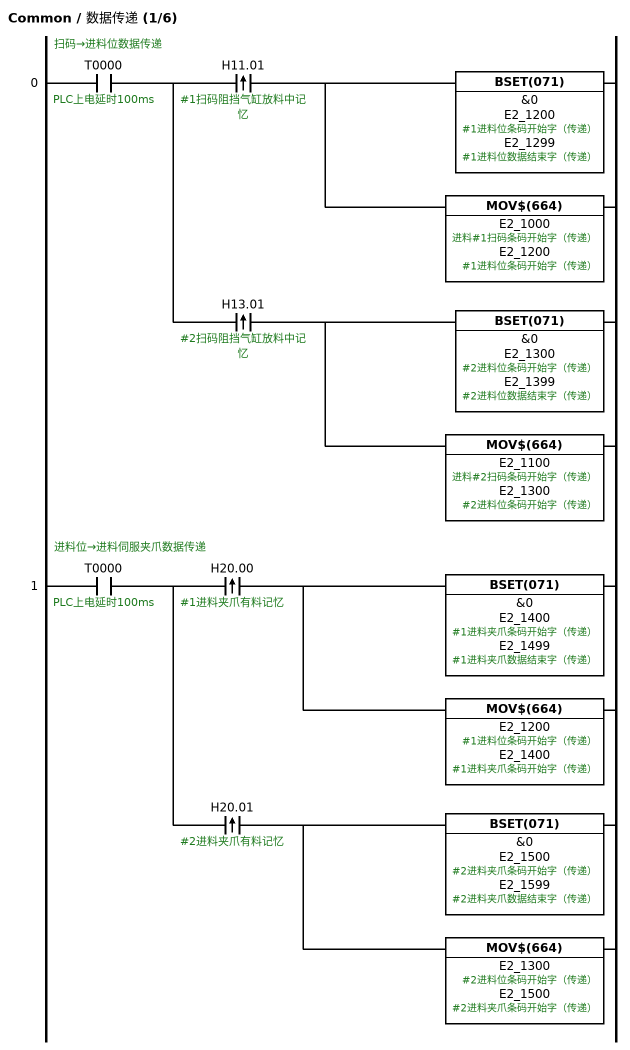
; [picture p528: Common / 数据传递, rungs 0-1]
; rung 0: 扫码→进料位数据传递
LD T0000  ; PLC上电延时100ms
OUT TR0
@AND H11.01  ; #1扫码阻挡气缸放料中记忆
BSET(071) &0 E2_1200 E2_1299  ; #1进料位条码开始字（传递）, #1进料位数据结束字（传递）
MOV$(664) E2_1000 E2_1200  ; 进料#1扫码条码开始字（传递）, #1进料位条码开始字（传递）
LD TR0
@AND H13.01  ; #2扫码阻挡气缸放料中记忆
BSET(071) &0 E2_1300 E2_1399  ; #2进料位条码开始字（传递）, #2进料位数据结束字（传递）
MOV$(664) E2_1100 E2_1300  ; 进料#2扫码条码开始字（传递）, #2进料位条码开始字（传递）
; rung 1: 进料位→进料伺服夹爪数据传递
LD T0000  ; PLC上电延时100ms
OUT TR0
@AND H20.00  ; #1进料夹爪有料记忆
BSET(071) &0 E2_1400 E2_1499  ; #1进料夹爪条码开始字（传递）, #1进料夹爪数据结束字（传递）
MOV$(664) E2_1200 E2_1400  ; #1进料位条码开始字（传递）, #1进料夹爪条码开始字（传递）
LD TR0
@AND H20.01  ; #2进料夹爪有料记忆
BSET(071) &0 E2_1500 E2_1599  ; #2进料夹爪条码开始字（传递）, #2进料夹爪数据结束字（传递）
MOV$(664) E2_1300 E2_1500  ; #2进料位条码开始字（传递）, #2进料夹爪条码开始字（传递）

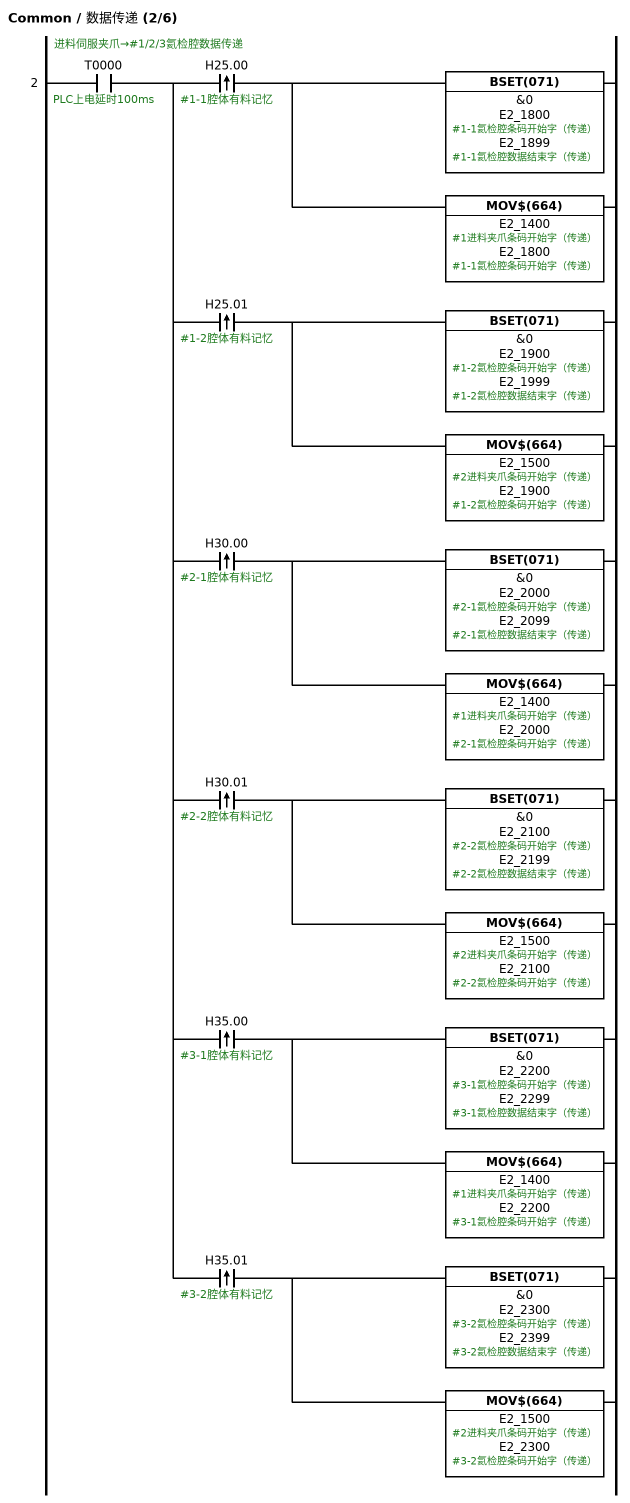
; rung 2: 进料伺服夹爪→#1/2/3氦检腔数据传递
LD T0000  ; PLC上电延时100ms
OUT TR0
@AND H25.00  ; #1-1腔体有料记忆
BSET(071) &0 E2_1800 E2_1899  ; #1-1氦检腔条码开始字（传递）, #1-1氦检腔数据结束字（传递）
MOV$(664) E2_1400 E2_1800  ; #1进料夹爪条码开始字（传递）, #1-1氦检腔条码开始字（传递）
LD TR0
@AND H25.01  ; #1-2腔体有料记忆
BSET(071) &0 E2_1900 E2_1999  ; #1-2氦检腔条码开始字（传递）, #1-2氦检腔数据结束字（传递）
MOV$(664) E2_1500 E2_1900  ; #2进料夹爪条码开始字（传递）, #1-2氦检腔条码开始字（传递）
LD TR0
@AND H30.00  ; #2-1腔体有料记忆
BSET(071) &0 E2_2000 E2_2099  ; #2-1氦检腔条码开始字（传递）, #2-1氦检腔数据结束字（传递）
MOV$(664) E2_1400 E2_2000  ; #1进料夹爪条码开始字（传递）, #2-1氦检腔条码开始字（传递）
LD TR0
@AND H30.01  ; #2-2腔体有料记忆
BSET(071) &0 E2_2100 E2_2199  ; #2-2氦检腔条码开始字（传递）, #2-2氦检腔数据结束字（传递）
MOV$(664) E2_1500 E2_2100  ; #2进料夹爪条码开始字（传递）, #2-2氦检腔条码开始字（传递）
LD TR0
@AND H35.00  ; #3-1腔体有料记忆
BSET(071) &0 E2_2200 E2_2299  ; #3-1氦检腔条码开始字（传递）, #3-1氦检腔数据结束字（传递）
MOV$(664) E2_1400 E2_2200  ; #1进料夹爪条码开始字（传递）, #3-1氦检腔条码开始字（传递）
LD TR0
@AND H35.01  ; #3-2腔体有料记忆
BSET(071) &0 E2_2300 E2_2399  ; #3-2氦检腔条码开始字（传递）, #3-2氦检腔数据结束字（传递）
MOV$(664) E2_1500 E2_2300  ; #2进料夹爪条码开始字（传递）, #3-2氦检腔条码开始字（传递）

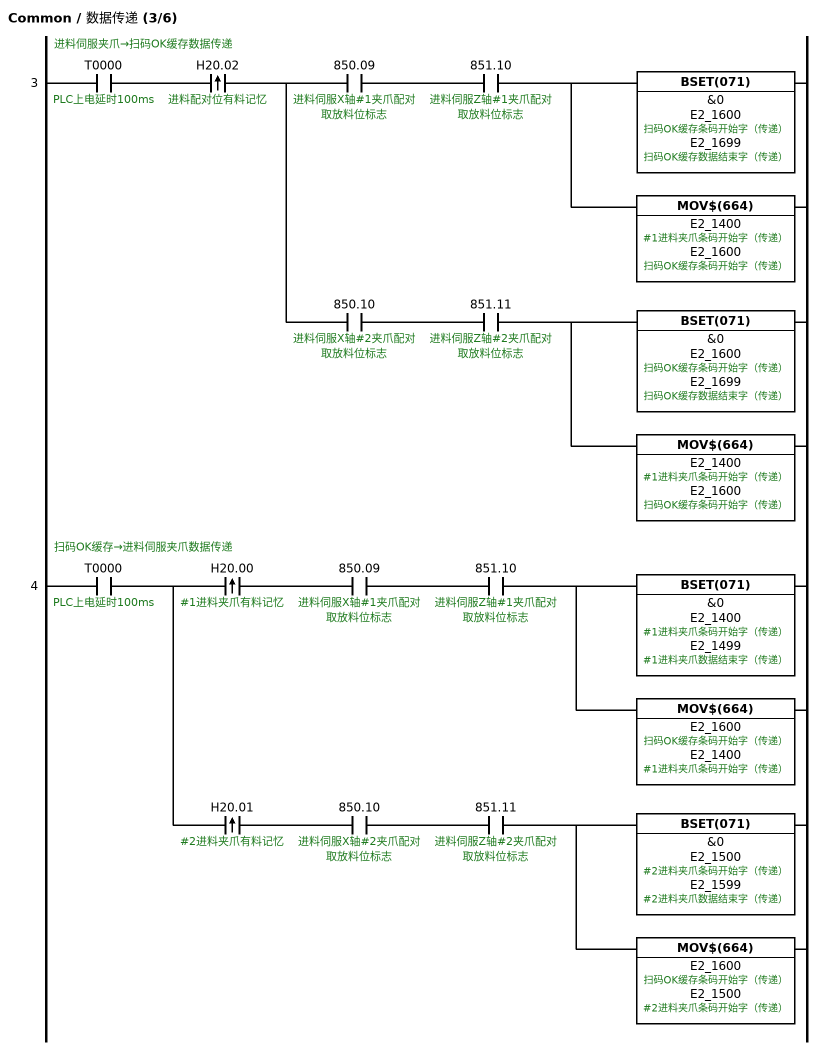
; rung 3: 进料伺服夹爪→扫码OK缓存数据传递
LD T0000  ; PLC上电延时100ms
@AND H20.02  ; 进料配对位有料记忆
OUT TR0
AND 850.09  ; 进料伺服X轴#1夹爪配对取放料位标志
AND 851.10  ; 进料伺服Z轴#1夹爪配对取放料位标志
BSET(071) &0 E2_1600 E2_1699  ; 扫码OK缓存条码开始字（传递）, 扫码OK缓存数据结束字（传递）
MOV$(664) E2_1400 E2_1600  ; #1进料夹爪条码开始字（传递）, 扫码OK缓存条码开始字（传递）
LD TR0
AND 850.10  ; 进料伺服X轴#2夹爪配对取放料位标志
AND 851.11  ; 进料伺服Z轴#2夹爪配对取放料位标志
BSET(071) &0 E2_1600 E2_1699  ; 扫码OK缓存条码开始字（传递）, 扫码OK缓存数据结束字（传递）
MOV$(664) E2_1400 E2_1600  ; #1进料夹爪条码开始字（传递）, 扫码OK缓存条码开始字（传递）
; rung 4: 扫码OK缓存→进料伺服夹爪数据传递
LD T0000  ; PLC上电延时100ms
OUT TR0
@AND H20.00  ; #1进料夹爪有料记忆
AND 850.09  ; 进料伺服X轴#1夹爪配对取放料位标志
AND 851.10  ; 进料伺服Z轴#1夹爪配对取放料位标志
BSET(071) &0 E2_1400 E2_1499  ; #1进料夹爪条码开始字（传递）, #1进料夹爪数据结束字（传递）
MOV$(664) E2_1600 E2_1400  ; 扫码OK缓存条码开始字（传递）, #1进料夹爪条码开始字（传递）
LD TR0
@AND H20.01  ; #2进料夹爪有料记忆
AND 850.10  ; 进料伺服X轴#2夹爪配对取放料位标志
AND 851.11  ; 进料伺服Z轴#2夹爪配对取放料位标志
BSET(071) &0 E2_1500 E2_1599  ; #2进料夹爪条码开始字（传递）, #2进料夹爪数据结束字（传递）
MOV$(664) E2_1600 E2_1500  ; 扫码OK缓存条码开始字（传递）, #2进料夹爪条码开始字（传递）

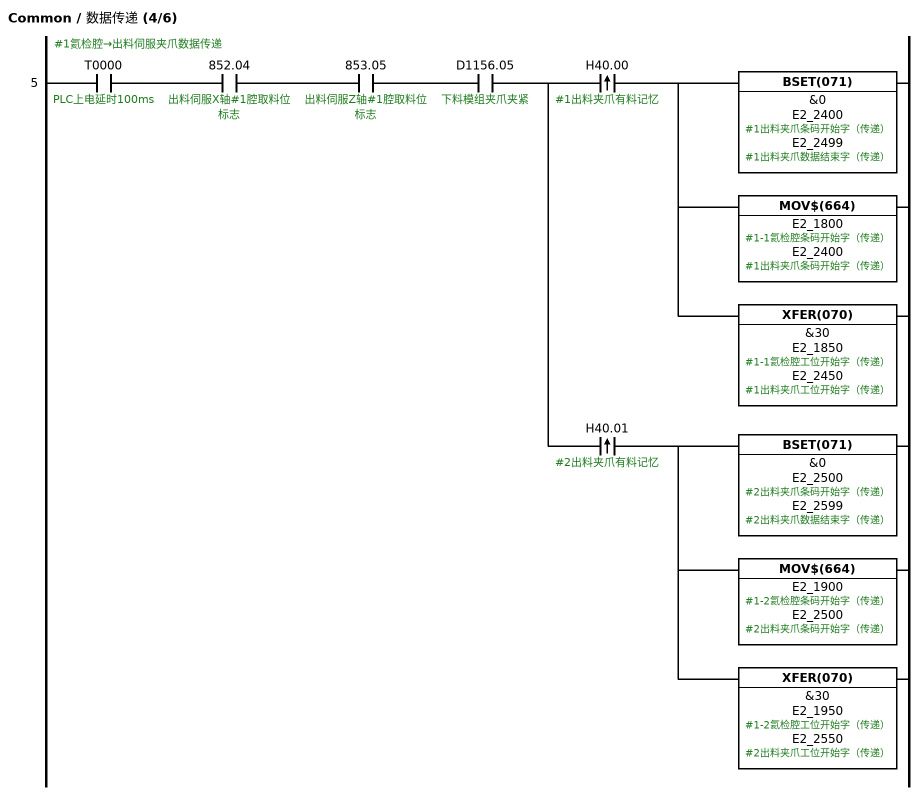
; rung 5: #1氦检腔→出料伺服夹爪数据传递
LD T0000  ; PLC上电延时100ms
AND 852.04  ; 出料伺服X轴#1腔取料位标志
AND 853.05  ; 出料伺服Z轴#1腔取料位标志
AND D1156.05  ; 下料模组夹爪夹紧
OUT TR0
@AND H40.00  ; #1出料夹爪有料记忆
BSET(071) &0 E2_2400 E2_2499  ; #1出料夹爪条码开始字（传递）, #1出料夹爪数据结束字（传递）
MOV$(664) E2_1800 E2_2400  ; #1-1氦检腔条码开始字（传递）, #1出料夹爪条码开始字（传递）
XFER(070) &30 E2_1850 E2_2450  ; #1-1氦检腔工位开始字（传递）, #1出料夹爪工位开始字（传递）
LD TR0
@AND H40.01  ; #2出料夹爪有料记忆
BSET(071) &0 E2_2500 E2_2599  ; #2出料夹爪条码开始字（传递）, #2出料夹爪数据结束字（传递）
MOV$(664) E2_1900 E2_2500  ; #1-2氦检腔条码开始字（传递）, #2出料夹爪条码开始字（传递）
XFER(070) &30 E2_1950 E2_2550  ; #1-2氦检腔工位开始字（传递）, #2出料夹爪工位开始字（传递）

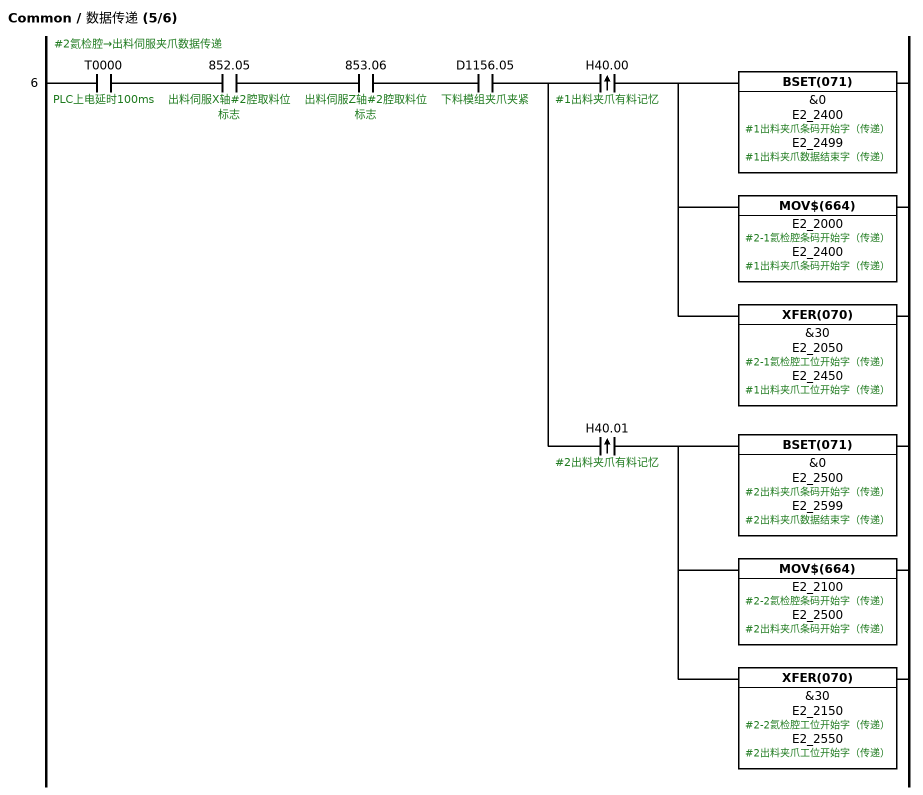
; rung 6: #2氦检腔→出料伺服夹爪数据传递
LD T0000  ; PLC上电延时100ms
AND 852.05  ; 出料伺服X轴#2腔取料位标志
AND 853.06  ; 出料伺服Z轴#2腔取料位标志
AND D1156.05  ; 下料模组夹爪夹紧
OUT TR0
@AND H40.00  ; #1出料夹爪有料记忆
BSET(071) &0 E2_2400 E2_2499  ; #1出料夹爪条码开始字（传递）, #1出料夹爪数据结束字（传递）
MOV$(664) E2_2000 E2_2400  ; #2-1氦检腔条码开始字（传递）, #1出料夹爪条码开始字（传递）
XFER(070) &30 E2_2050 E2_2450  ; #2-1氦检腔工位开始字（传递）, #1出料夹爪工位开始字（传递）
LD TR0
@AND H40.01  ; #2出料夹爪有料记忆
BSET(071) &0 E2_2500 E2_2599  ; #2出料夹爪条码开始字（传递）, #2出料夹爪数据结束字（传递）
MOV$(664) E2_2100 E2_2500  ; #2-2氦检腔条码开始字（传递）, #2出料夹爪条码开始字（传递）
XFER(070) &30 E2_2150 E2_2550  ; #2-2氦检腔工位开始字（传递）, #2出料夹爪工位开始字（传递）

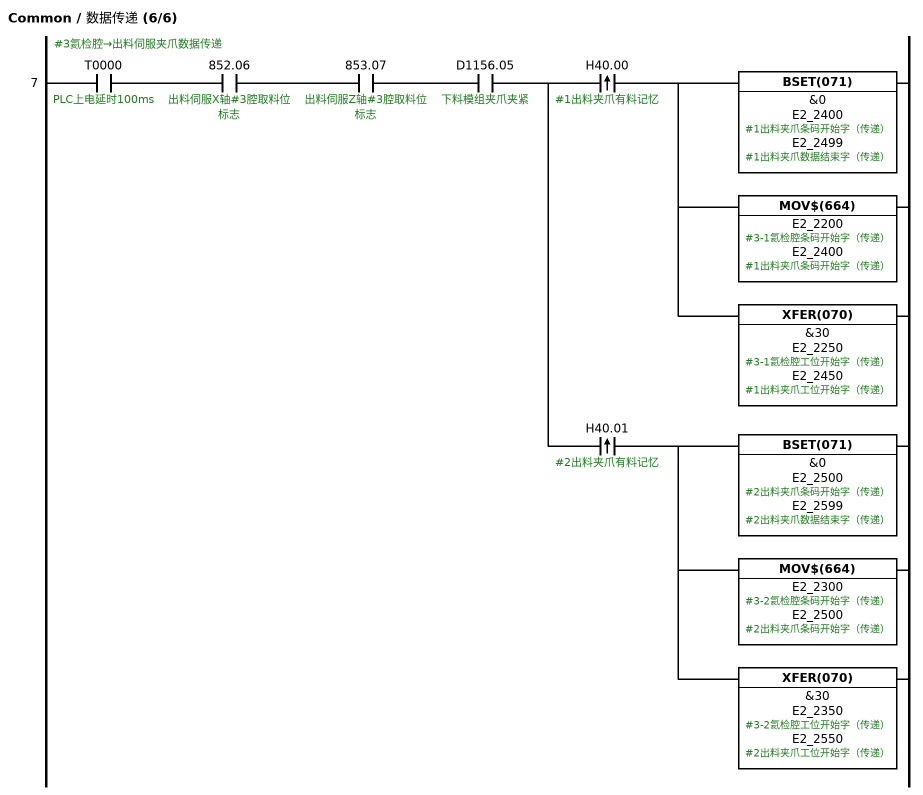
; rung 7: #3氦检腔→出料伺服夹爪数据传递
LD T0000  ; PLC上电延时100ms
AND 852.06  ; 出料伺服X轴#3腔取料位标志
AND 853.07  ; 出料伺服Z轴#3腔取料位标志
AND D1156.05  ; 下料模组夹爪夹紧
OUT TR0
@AND H40.00  ; #1出料夹爪有料记忆
BSET(071) &0 E2_2400 E2_2499  ; #1出料夹爪条码开始字（传递）, #1出料夹爪数据结束字（传递）
MOV$(664) E2_2200 E2_2400  ; #3-1氦检腔条码开始字（传递）, #1出料夹爪条码开始字（传递）
XFER(070) &30 E2_2250 E2_2450  ; #3-1氦检腔工位开始字（传递）, #1出料夹爪工位开始字（传递）
LD TR0
@AND H40.01  ; #2出料夹爪有料记忆
BSET(071) &0 E2_2500 E2_2599  ; #2出料夹爪条码开始字（传递）, #2出料夹爪数据结束字（传递）
MOV$(664) E2_2300 E2_2500  ; #3-2氦检腔条码开始字（传递）, #2出料夹爪条码开始字（传递）
XFER(070) &30 E2_2350 E2_2550  ; #3-2氦检腔工位开始字（传递）, #2出料夹爪工位开始字（传递）

### Section 数据处理

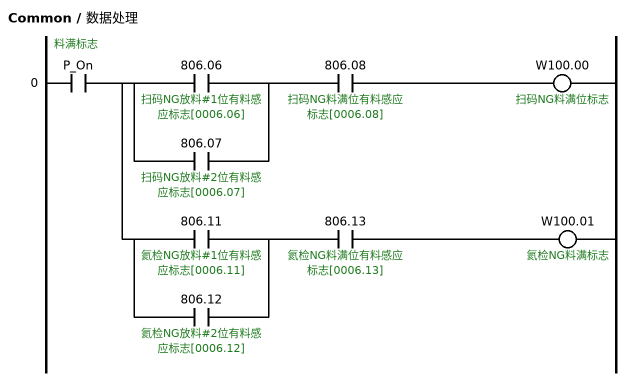
; rung 0: 料满标志
LD P_On
OUT TR0
LD 806.06  ; 扫码NG放料#1位有料感应标志[0006.06]
OR 806.07  ; 扫码NG放料#2位有料感应标志[0006.07]
ANDLD
AND 806.08  ; 扫码NG料满位有料感应标志[0006.08]
OUT W100.00  ; 扫码NG料满位标志
LD TR0
LD 806.11  ; 氦检NG放料#1位有料感应标志[0006.11]
OR 806.12  ; 氦检NG放料#2位有料感应标志[0006.12]
ANDLD
AND 806.13  ; 氦检NG料满位有料感应标志[0006.13]
OUT W100.01  ; 氦检NG料满标志

### Section 报警

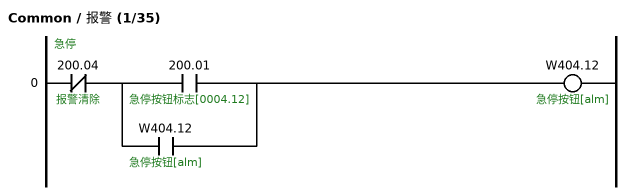
; rung 0: 急停
LDNOT 200.04  ; 报警清除
LD 200.01  ; 急停按钮标志[0004.12]
OR W404.12  ; 急停按钮[alm]
ANDLD
OUT W404.12  ; 急停按钮[alm]

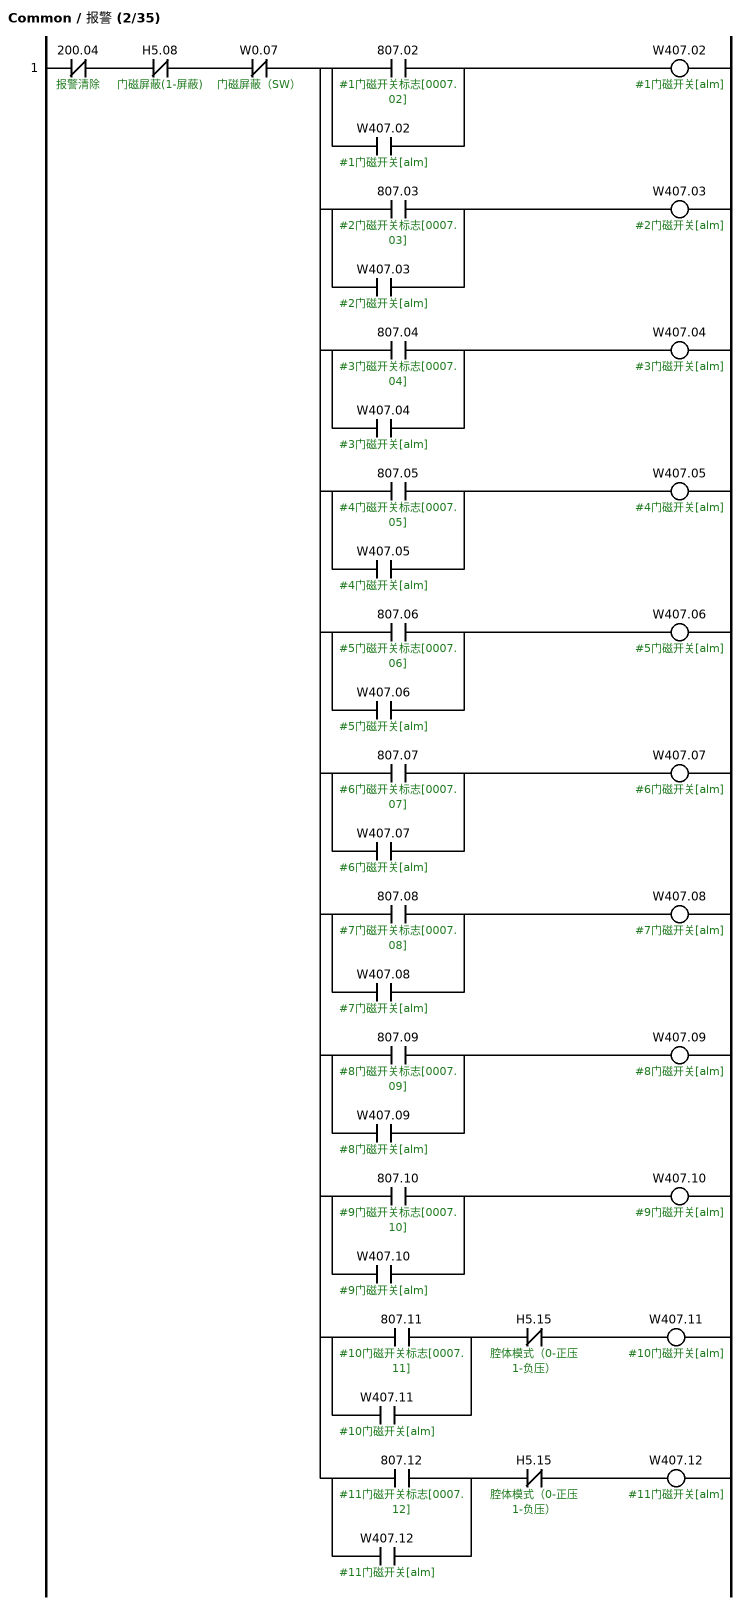
; rung 1
LDNOT 200.04  ; 报警清除
ANDNOT H5.08  ; 门磁屏蔽(1-屏蔽)
ANDNOT W0.07  ; 门磁屏蔽（SW）
OUT TR0
LD 807.02  ; #1门磁开关标志[0007.02]
OR W407.02  ; #1门磁开关[alm]
ANDLD
OUT W407.02  ; #1门磁开关[alm]
LD TR0
LD 807.03  ; #2门磁开关标志[0007.03]
OR W407.03  ; #2门磁开关[alm]
ANDLD
OUT W407.03  ; #2门磁开关[alm]
LD TR0
LD 807.04  ; #3门磁开关标志[0007.04]
OR W407.04  ; #3门磁开关[alm]
ANDLD
OUT W407.04  ; #3门磁开关[alm]
LD TR0
LD 807.05  ; #4门磁开关标志[0007.05]
OR W407.05  ; #4门磁开关[alm]
ANDLD
OUT W407.05  ; #4门磁开关[alm]
LD TR0
LD 807.06  ; #5门磁开关标志[0007.06]
OR W407.06  ; #5门磁开关[alm]
ANDLD
OUT W407.06  ; #5门磁开关[alm]
LD TR0
LD 807.07  ; #6门磁开关标志[0007.07]
OR W407.07  ; #6门磁开关[alm]
ANDLD
OUT W407.07  ; #6门磁开关[alm]
LD TR0
LD 807.08  ; #7门磁开关标志[0007.08]
OR W407.08  ; #7门磁开关[alm]
ANDLD
OUT W407.08  ; #7门磁开关[alm]
LD TR0
LD 807.09  ; #8门磁开关标志[0007.09]
OR W407.09  ; #8门磁开关[alm]
ANDLD
OUT W407.09  ; #8门磁开关[alm]
LD TR0
LD 807.10  ; #9门磁开关标志[0007.10]
OR W407.10  ; #9门磁开关[alm]
ANDLD
OUT W407.10  ; #9门磁开关[alm]
LD TR0
LD 807.11  ; #10门磁开关标志[0007.11]
OR W407.11  ; #10门磁开关[alm]
ANDLD
ANDNOT H5.15  ; 腔体模式（0-正压 1-负压）
OUT W407.11  ; #10门磁开关[alm]
LD TR0
LD 807.12  ; #11门磁开关标志[0007.12]
OR W407.12  ; #11门磁开关[alm]
ANDLD
ANDNOT H5.15  ; 腔体模式（0-正压 1-负压）
OUT W407.12  ; #11门磁开关[alm]

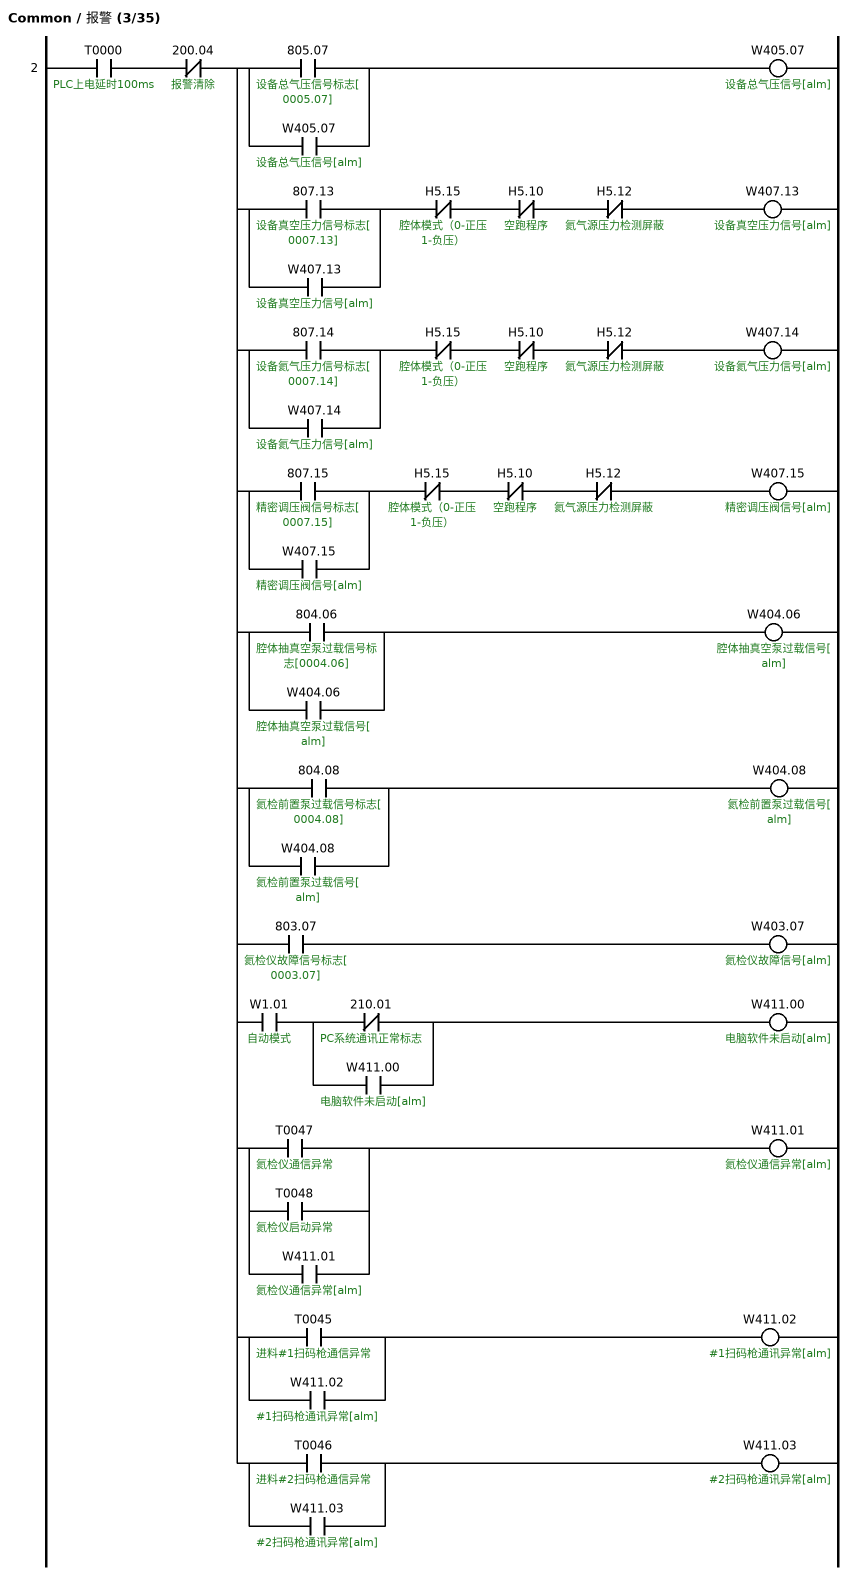
; rung 2
LD T0000  ; PLC上电延时100ms
ANDNOT 200.04  ; 报警清除
OUT TR0
LD 805.07  ; 设备总气压信号标志[0005.07]
OR W405.07  ; 设备总气压信号[alm]
ANDLD
OUT W405.07  ; 设备总气压信号[alm]
LD TR0
LD 807.13  ; 设备真空压力信号标志[0007.13]
OR W407.13  ; 设备真空压力信号[alm]
ANDLD
ANDNOT H5.15  ; 腔体模式（0-正压 1-负压）
ANDNOT H5.10  ; 空跑程序
ANDNOT H5.12  ; 氦气源压力检测屏蔽
OUT W407.13  ; 设备真空压力信号[alm]
LD TR0
LD 807.14  ; 设备氦气压力信号标志[0007.14]
OR W407.14  ; 设备氦气压力信号[alm]
ANDLD
ANDNOT H5.15  ; 腔体模式（0-正压 1-负压）
ANDNOT H5.10  ; 空跑程序
ANDNOT H5.12  ; 氦气源压力检测屏蔽
OUT W407.14  ; 设备氦气压力信号[alm]
LD TR0
LD 807.15  ; 精密调压阀信号标志[0007.15]
OR W407.15  ; 精密调压阀信号[alm]
ANDLD
ANDNOT H5.15  ; 腔体模式（0-正压 1-负压）
ANDNOT H5.10  ; 空跑程序
ANDNOT H5.12  ; 氦气源压力检测屏蔽
OUT W407.15  ; 精密调压阀信号[alm]
LD TR0
LD 804.06  ; 腔体抽真空泵过载信号标志[0004.06]
OR W404.06  ; 腔体抽真空泵过载信号[alm]
ANDLD
OUT W404.06  ; 腔体抽真空泵过载信号[alm]
LD TR0
LD 804.08  ; 氦检前置泵过载信号标志[0004.08]
OR W404.08  ; 氦检前置泵过载信号[alm]
ANDLD
OUT W404.08  ; 氦检前置泵过载信号[alm]
LD TR0
AND 803.07  ; 氦检仪故障信号标志[0003.07]
OUT W403.07  ; 氦检仪故障信号[alm]
LD TR0
AND W1.01  ; 自动模式
LDNOT 210.01  ; PC系统通讯正常标志
OR W411.00  ; 电脑软件未启动[alm]
ANDLD
OUT W411.00  ; 电脑软件未启动[alm]
LD TR0
LD T0047  ; 氦检仪通信异常
OR T0048  ; 氦检仪启动异常
OR W411.01  ; 氦检仪通信异常[alm]
ANDLD
OUT W411.01  ; 氦检仪通信异常[alm]
LD TR0
LD T0045  ; 进料#1扫码枪通信异常
OR W411.02  ; #1扫码枪通讯异常[alm]
ANDLD
OUT W411.02  ; #1扫码枪通讯异常[alm]
LD TR0
LD T0046  ; 进料#2扫码枪通信异常
OR W411.03  ; #2扫码枪通讯异常[alm]
ANDLD
OUT W411.03  ; #2扫码枪通讯异常[alm]

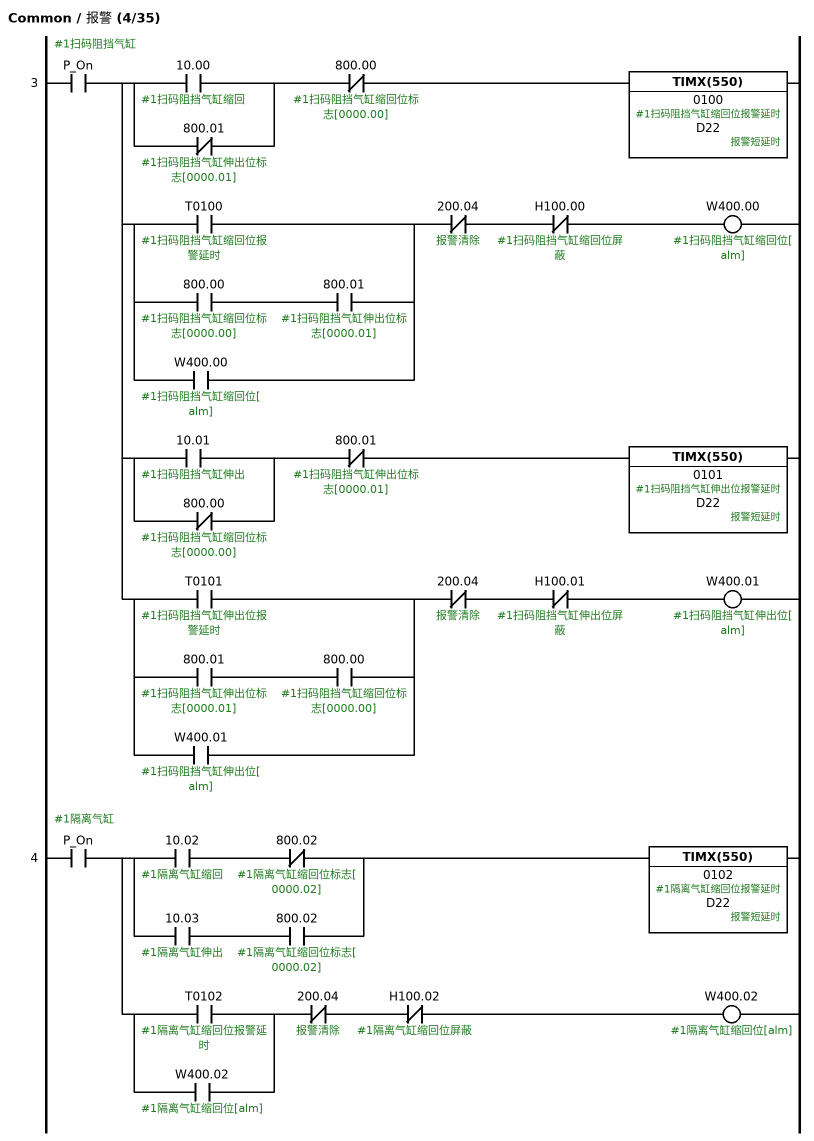
; rung 3: #1扫码阻挡气缸
LD P_On
OUT TR0
LD 10.00  ; #1扫码阻挡气缸缩回
ORNOT 800.01  ; #1扫码阻挡气缸伸出位标志[0000.01]
ANDLD
ANDNOT 800.00  ; #1扫码阻挡气缸缩回位标志[0000.00]
TIMX(550) 0100 D22  ; 报警短延时, #1扫码阻挡气缸缩回位报警延时
LD TR0
LD T0100  ; #1扫码阻挡气缸缩回位报警延时
LD 800.00  ; #1扫码阻挡气缸缩回位标志[0000.00]
AND 800.01  ; #1扫码阻挡气缸伸出位标志[0000.01]
ORLD
OR W400.00  ; #1扫码阻挡气缸缩回位[alm]
ANDLD
ANDNOT 200.04  ; 报警清除
ANDNOT H100.00  ; #1扫码阻挡气缸缩回位屏蔽
OUT W400.00  ; #1扫码阻挡气缸缩回位[alm]
LD TR0
LD 10.01  ; #1扫码阻挡气缸伸出
ORNOT 800.00  ; #1扫码阻挡气缸缩回位标志[0000.00]
ANDLD
ANDNOT 800.01  ; #1扫码阻挡气缸伸出位标志[0000.01]
TIMX(550) 0101 D22  ; 报警短延时, #1扫码阻挡气缸伸出位报警延时
LD TR0
LD T0101  ; #1扫码阻挡气缸伸出位报警延时
LD 800.01  ; #1扫码阻挡气缸伸出位标志[0000.01]
AND 800.00  ; #1扫码阻挡气缸缩回位标志[0000.00]
ORLD
OR W400.01  ; #1扫码阻挡气缸伸出位[alm]
ANDLD
ANDNOT 200.04  ; 报警清除
ANDNOT H100.01  ; #1扫码阻挡气缸伸出位屏蔽
OUT W400.01  ; #1扫码阻挡气缸伸出位[alm]
; rung 4: #1隔离气缸
LD P_On
OUT TR0
LD 10.02  ; #1隔离气缸缩回
ANDNOT 800.02  ; #1隔离气缸缩回位标志[0000.02]
LD 10.03  ; #1隔离气缸伸出
AND 800.02  ; #1隔离气缸缩回位标志[0000.02]
ORLD
ANDLD
TIMX(550) 0102 D22  ; 报警短延时, #1隔离气缸缩回位报警延时
LD TR0
LD T0102  ; #1隔离气缸缩回位报警延时
OR W400.02  ; #1隔离气缸缩回位[alm]
ANDLD
ANDNOT 200.04  ; 报警清除
ANDNOT H100.02  ; #1隔离气缸缩回位屏蔽
OUT W400.02  ; #1隔离气缸缩回位[alm]

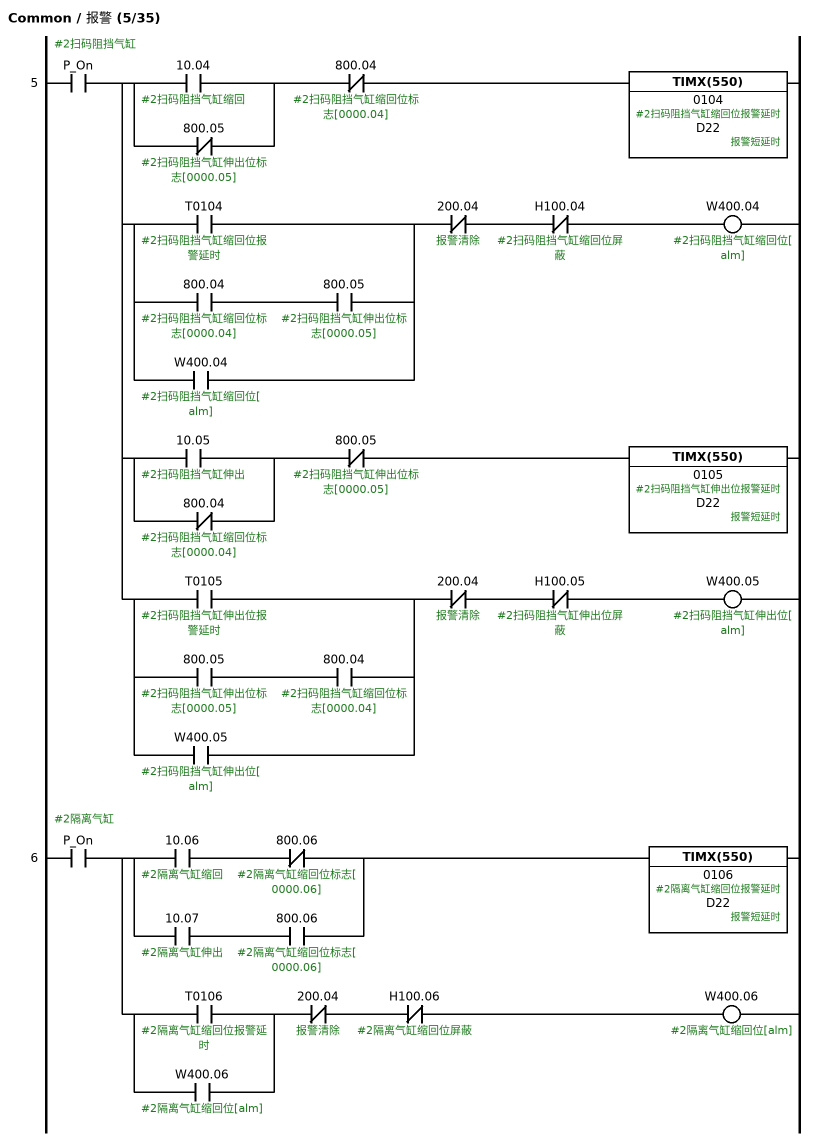
; rung 5: #2扫码阻挡气缸
LD P_On
OUT TR0
LD 10.04  ; #2扫码阻挡气缸缩回
ORNOT 800.05  ; #2扫码阻挡气缸伸出位标志[0000.05]
ANDLD
ANDNOT 800.04  ; #2扫码阻挡气缸缩回位标志[0000.04]
TIMX(550) 0104 D22  ; 报警短延时, #2扫码阻挡气缸缩回位报警延时
LD TR0
LD T0104  ; #2扫码阻挡气缸缩回位报警延时
LD 800.04  ; #2扫码阻挡气缸缩回位标志[0000.04]
AND 800.05  ; #2扫码阻挡气缸伸出位标志[0000.05]
ORLD
OR W400.04  ; #2扫码阻挡气缸缩回位[alm]
ANDLD
ANDNOT 200.04  ; 报警清除
ANDNOT H100.04  ; #2扫码阻挡气缸缩回位屏蔽
OUT W400.04  ; #2扫码阻挡气缸缩回位[alm]
LD TR0
LD 10.05  ; #2扫码阻挡气缸伸出
ORNOT 800.04  ; #2扫码阻挡气缸缩回位标志[0000.04]
ANDLD
ANDNOT 800.05  ; #2扫码阻挡气缸伸出位标志[0000.05]
TIMX(550) 0105 D22  ; 报警短延时, #2扫码阻挡气缸伸出位报警延时
LD TR0
LD T0105  ; #2扫码阻挡气缸伸出位报警延时
LD 800.05  ; #2扫码阻挡气缸伸出位标志[0000.05]
AND 800.04  ; #2扫码阻挡气缸缩回位标志[0000.04]
ORLD
OR W400.05  ; #2扫码阻挡气缸伸出位[alm]
ANDLD
ANDNOT 200.04  ; 报警清除
ANDNOT H100.05  ; #2扫码阻挡气缸伸出位屏蔽
OUT W400.05  ; #2扫码阻挡气缸伸出位[alm]
; rung 6: #2隔离气缸
LD P_On
OUT TR0
LD 10.06  ; #2隔离气缸缩回
ANDNOT 800.06  ; #2隔离气缸缩回位标志[0000.06]
LD 10.07  ; #2隔离气缸伸出
AND 800.06  ; #2隔离气缸缩回位标志[0000.06]
ORLD
ANDLD
TIMX(550) 0106 D22  ; 报警短延时, #2隔离气缸缩回位报警延时
LD TR0
LD T0106  ; #2隔离气缸缩回位报警延时
OR W400.06  ; #2隔离气缸缩回位[alm]
ANDLD
ANDNOT 200.04  ; 报警清除
ANDNOT H100.06  ; #2隔离气缸缩回位屏蔽
OUT W400.06  ; #2隔离气缸缩回位[alm]

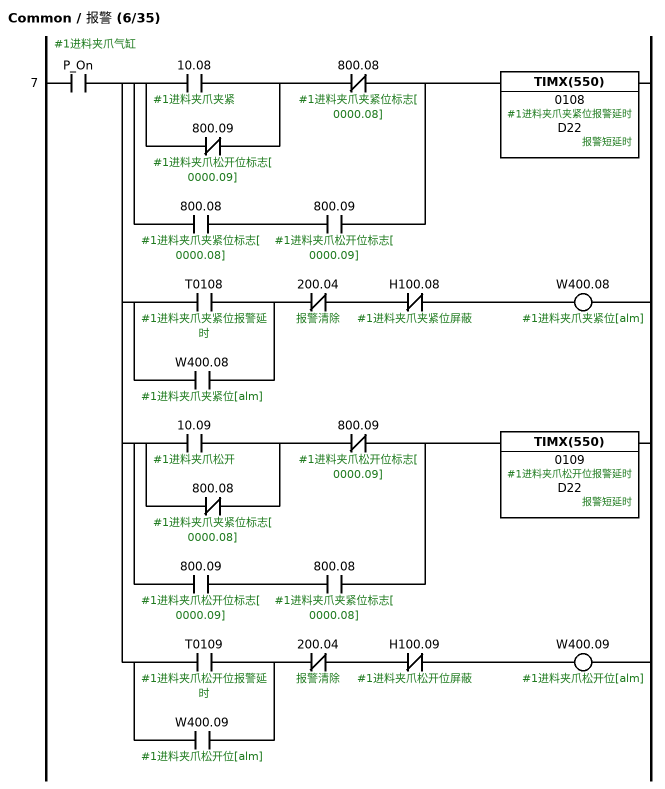
; rung 7: #1进料夹爪气缸
LD P_On
OUT TR0
LD 10.08  ; #1进料夹爪夹紧
ORNOT 800.09  ; #1进料夹爪松开位标志[0000.09]
ANDNOT 800.08  ; #1进料夹爪夹紧位标志[0000.08]
LD 800.08  ; #1进料夹爪夹紧位标志[0000.08]
AND 800.09  ; #1进料夹爪松开位标志[0000.09]
ORLD
ANDLD
TIMX(550) 0108 D22  ; 报警短延时, #1进料夹爪夹紧位报警延时
LD TR0
LD T0108  ; #1进料夹爪夹紧位报警延时
OR W400.08  ; #1进料夹爪夹紧位[alm]
ANDLD
ANDNOT 200.04  ; 报警清除
ANDNOT H100.08  ; #1进料夹爪夹紧位屏蔽
OUT W400.08  ; #1进料夹爪夹紧位[alm]
LD TR0
LD 10.09  ; #1进料夹爪松开
ORNOT 800.08  ; #1进料夹爪夹紧位标志[0000.08]
ANDNOT 800.09  ; #1进料夹爪松开位标志[0000.09]
LD 800.09  ; #1进料夹爪松开位标志[0000.09]
AND 800.08  ; #1进料夹爪夹紧位标志[0000.08]
ORLD
ANDLD
TIMX(550) 0109 D22  ; 报警短延时, #1进料夹爪松开位报警延时
LD TR0
LD T0109  ; #1进料夹爪松开位报警延时
OR W400.09  ; #1进料夹爪松开位[alm]
ANDLD
ANDNOT 200.04  ; 报警清除
ANDNOT H100.09  ; #1进料夹爪松开位屏蔽
OUT W400.09  ; #1进料夹爪松开位[alm]

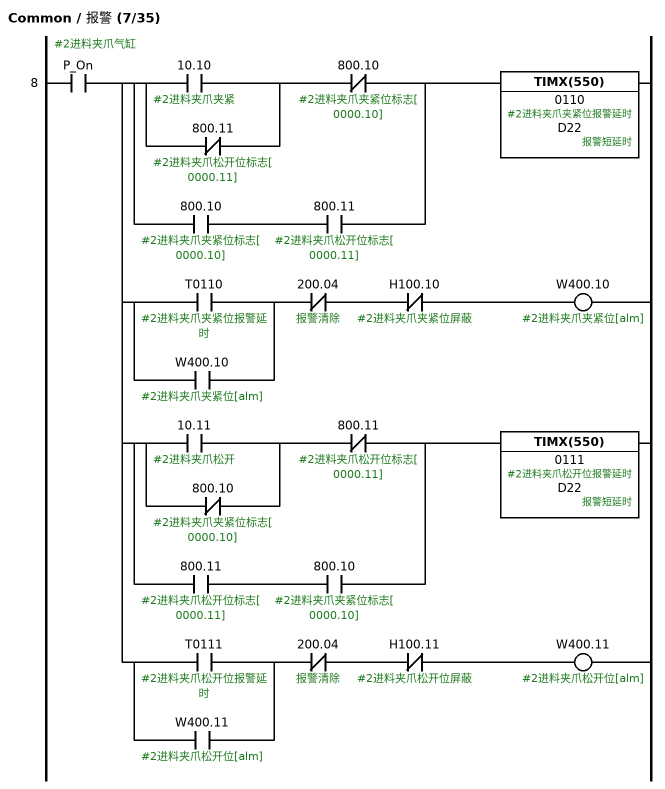
; rung 8: #2进料夹爪气缸
LD P_On
OUT TR0
LD 10.10  ; #2进料夹爪夹紧
ORNOT 800.11  ; #2进料夹爪松开位标志[0000.11]
ANDNOT 800.10  ; #2进料夹爪夹紧位标志[0000.10]
LD 800.10  ; #2进料夹爪夹紧位标志[0000.10]
AND 800.11  ; #2进料夹爪松开位标志[0000.11]
ORLD
ANDLD
TIMX(550) 0110 D22  ; 报警短延时, #2进料夹爪夹紧位报警延时
LD TR0
LD T0110  ; #2进料夹爪夹紧位报警延时
OR W400.10  ; #2进料夹爪夹紧位[alm]
ANDLD
ANDNOT 200.04  ; 报警清除
ANDNOT H100.10  ; #2进料夹爪夹紧位屏蔽
OUT W400.10  ; #2进料夹爪夹紧位[alm]
LD TR0
LD 10.11  ; #2进料夹爪松开
ORNOT 800.10  ; #2进料夹爪夹紧位标志[0000.10]
ANDNOT 800.11  ; #2进料夹爪松开位标志[0000.11]
LD 800.11  ; #2进料夹爪松开位标志[0000.11]
AND 800.10  ; #2进料夹爪夹紧位标志[0000.10]
ORLD
ANDLD
TIMX(550) 0111 D22  ; 报警短延时, #2进料夹爪松开位报警延时
LD TR0
LD T0111  ; #2进料夹爪松开位报警延时
OR W400.11  ; #2进料夹爪松开位[alm]
ANDLD
ANDNOT 200.04  ; 报警清除
ANDNOT H100.11  ; #2进料夹爪松开位屏蔽
OUT W400.11  ; #2进料夹爪松开位[alm]

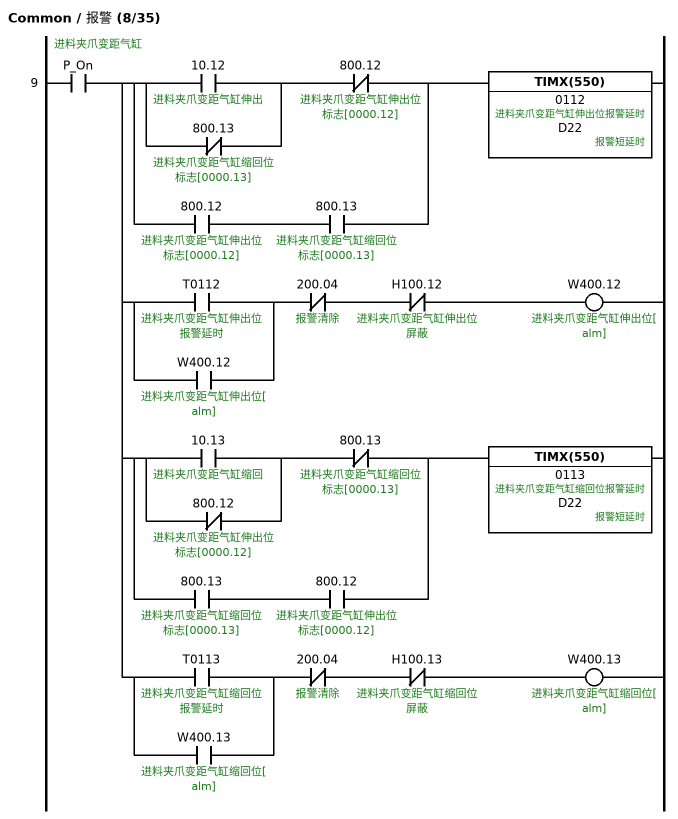
; rung 9: 进料夹爪变距气缸
LD P_On
OUT TR0
LD 10.12  ; 进料夹爪变距气缸伸出
ORNOT 800.13  ; 进料夹爪变距气缸缩回位标志[0000.13]
ANDNOT 800.12  ; 进料夹爪变距气缸伸出位标志[0000.12]
LD 800.12  ; 进料夹爪变距气缸伸出位标志[0000.12]
AND 800.13  ; 进料夹爪变距气缸缩回位标志[0000.13]
ORLD
ANDLD
TIMX(550) 0112 D22  ; 报警短延时, 进料夹爪变距气缸伸出位报警延时
LD TR0
LD T0112  ; 进料夹爪变距气缸伸出位报警延时
OR W400.12  ; 进料夹爪变距气缸伸出位[alm]
ANDLD
ANDNOT 200.04  ; 报警清除
ANDNOT H100.12  ; 进料夹爪变距气缸伸出位屏蔽
OUT W400.12  ; 进料夹爪变距气缸伸出位[alm]
LD TR0
LD 10.13  ; 进料夹爪变距气缸缩回
ORNOT 800.12  ; 进料夹爪变距气缸伸出位标志[0000.12]
ANDNOT 800.13  ; 进料夹爪变距气缸缩回位标志[0000.13]
LD 800.13  ; 进料夹爪变距气缸缩回位标志[0000.13]
AND 800.12  ; 进料夹爪变距气缸伸出位标志[0000.12]
ORLD
ANDLD
TIMX(550) 0113 D22  ; 报警短延时, 进料夹爪变距气缸缩回位报警延时
LD TR0
LD T0113  ; 进料夹爪变距气缸缩回位报警延时
OR W400.13  ; 进料夹爪变距气缸缩回位[alm]
ANDLD
ANDNOT 200.04  ; 报警清除
ANDNOT H100.13  ; 进料夹爪变距气缸缩回位屏蔽
OUT W400.13  ; 进料夹爪变距气缸缩回位[alm]

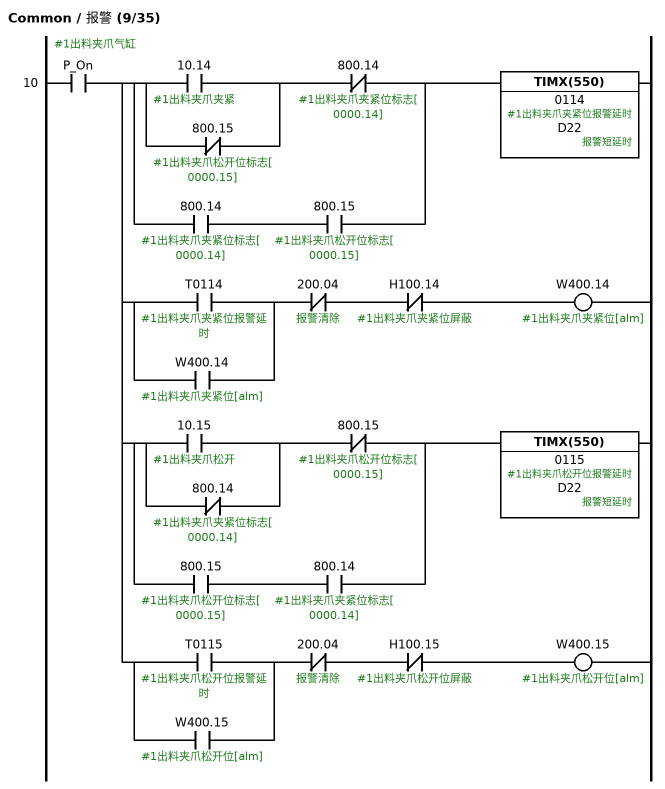
; rung 10: #1出料夹爪气缸
LD P_On
OUT TR0
LD 10.14  ; #1出料夹爪夹紧
ORNOT 800.15  ; #1出料夹爪松开位标志[0000.15]
ANDNOT 800.14  ; #1出料夹爪夹紧位标志[0000.14]
LD 800.14  ; #1出料夹爪夹紧位标志[0000.14]
AND 800.15  ; #1出料夹爪松开位标志[0000.15]
ORLD
ANDLD
TIMX(550) 0114 D22  ; 报警短延时, #1出料夹爪夹紧位报警延时
LD TR0
LD T0114  ; #1出料夹爪夹紧位报警延时
OR W400.14  ; #1出料夹爪夹紧位[alm]
ANDLD
ANDNOT 200.04  ; 报警清除
ANDNOT H100.14  ; #1出料夹爪夹紧位屏蔽
OUT W400.14  ; #1出料夹爪夹紧位[alm]
LD TR0
LD 10.15  ; #1出料夹爪松开
ORNOT 800.14  ; #1出料夹爪夹紧位标志[0000.14]
ANDNOT 800.15  ; #1出料夹爪松开位标志[0000.15]
LD 800.15  ; #1出料夹爪松开位标志[0000.15]
AND 800.14  ; #1出料夹爪夹紧位标志[0000.14]
ORLD
ANDLD
TIMX(550) 0115 D22  ; 报警短延时, #1出料夹爪松开位报警延时
LD TR0
LD T0115  ; #1出料夹爪松开位报警延时
OR W400.15  ; #1出料夹爪松开位[alm]
ANDLD
ANDNOT 200.04  ; 报警清除
ANDNOT H100.15  ; #1出料夹爪松开位屏蔽
OUT W400.15  ; #1出料夹爪松开位[alm]

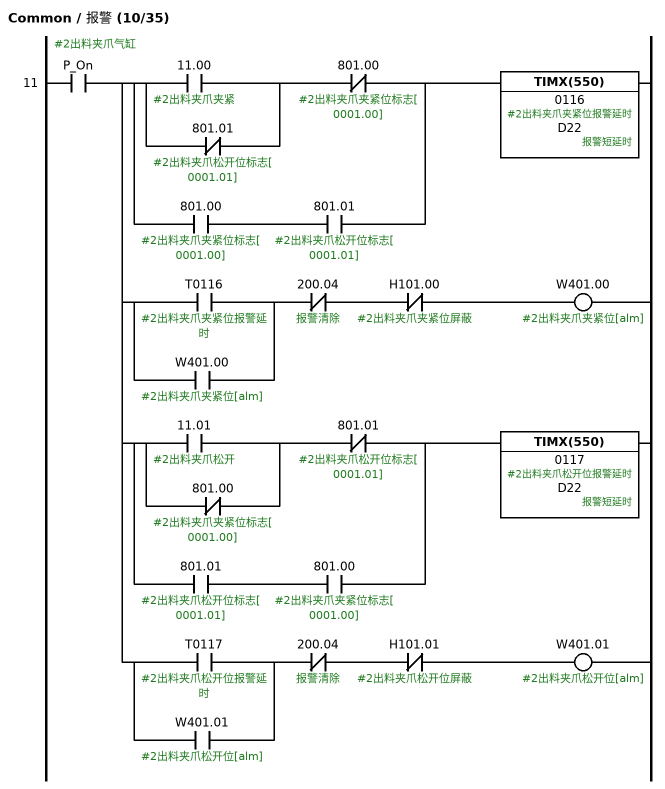
; rung 11: #2出料夹爪气缸
LD P_On
OUT TR0
LD 11.00  ; #2出料夹爪夹紧
ORNOT 801.01  ; #2出料夹爪松开位标志[0001.01]
ANDNOT 801.00  ; #2出料夹爪夹紧位标志[0001.00]
LD 801.00  ; #2出料夹爪夹紧位标志[0001.00]
AND 801.01  ; #2出料夹爪松开位标志[0001.01]
ORLD
ANDLD
TIMX(550) 0116 D22  ; 报警短延时, #2出料夹爪夹紧位报警延时
LD TR0
LD T0116  ; #2出料夹爪夹紧位报警延时
OR W401.00  ; #2出料夹爪夹紧位[alm]
ANDLD
ANDNOT 200.04  ; 报警清除
ANDNOT H101.00  ; #2出料夹爪夹紧位屏蔽
OUT W401.00  ; #2出料夹爪夹紧位[alm]
LD TR0
LD 11.01  ; #2出料夹爪松开
ORNOT 801.00  ; #2出料夹爪夹紧位标志[0001.00]
ANDNOT 801.01  ; #2出料夹爪松开位标志[0001.01]
LD 801.01  ; #2出料夹爪松开位标志[0001.01]
AND 801.00  ; #2出料夹爪夹紧位标志[0001.00]
ORLD
ANDLD
TIMX(550) 0117 D22  ; 报警短延时, #2出料夹爪松开位报警延时
LD TR0
LD T0117  ; #2出料夹爪松开位报警延时
OR W401.01  ; #2出料夹爪松开位[alm]
ANDLD
ANDNOT 200.04  ; 报警清除
ANDNOT H101.01  ; #2出料夹爪松开位屏蔽
OUT W401.01  ; #2出料夹爪松开位[alm]

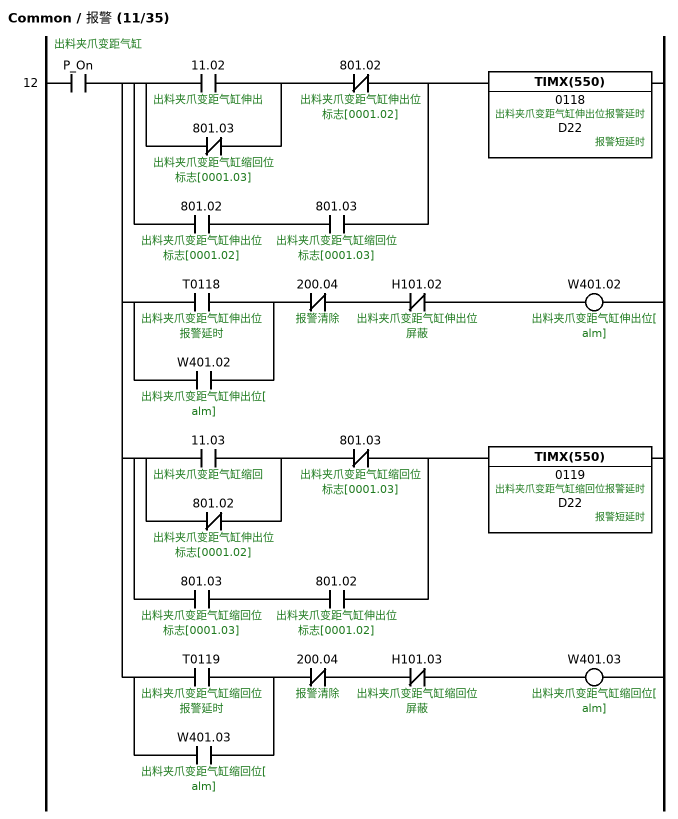
; rung 12: 出料夹爪变距气缸
LD P_On
OUT TR0
LD 11.02  ; 出料夹爪变距气缸伸出
ORNOT 801.03  ; 出料夹爪变距气缸缩回位标志[0001.03]
ANDNOT 801.02  ; 出料夹爪变距气缸伸出位标志[0001.02]
LD 801.02  ; 出料夹爪变距气缸伸出位标志[0001.02]
AND 801.03  ; 出料夹爪变距气缸缩回位标志[0001.03]
ORLD
ANDLD
TIMX(550) 0118 D22  ; 报警短延时, 出料夹爪变距气缸伸出位报警延时
LD TR0
LD T0118  ; 出料夹爪变距气缸伸出位报警延时
OR W401.02  ; 出料夹爪变距气缸伸出位[alm]
ANDLD
ANDNOT 200.04  ; 报警清除
ANDNOT H101.02  ; 出料夹爪变距气缸伸出位屏蔽
OUT W401.02  ; 出料夹爪变距气缸伸出位[alm]
LD TR0
LD 11.03  ; 出料夹爪变距气缸缩回
ORNOT 801.02  ; 出料夹爪变距气缸伸出位标志[0001.02]
ANDNOT 801.03  ; 出料夹爪变距气缸缩回位标志[0001.03]
LD 801.03  ; 出料夹爪变距气缸缩回位标志[0001.03]
AND 801.02  ; 出料夹爪变距气缸伸出位标志[0001.02]
ORLD
ANDLD
TIMX(550) 0119 D22  ; 报警短延时, 出料夹爪变距气缸缩回位报警延时
LD TR0
LD T0119  ; 出料夹爪变距气缸缩回位报警延时
OR W401.03  ; 出料夹爪变距气缸缩回位[alm]
ANDLD
ANDNOT 200.04  ; 报警清除
ANDNOT H101.03  ; 出料夹爪变距气缸缩回位屏蔽
OUT W401.03  ; 出料夹爪变距气缸缩回位[alm]

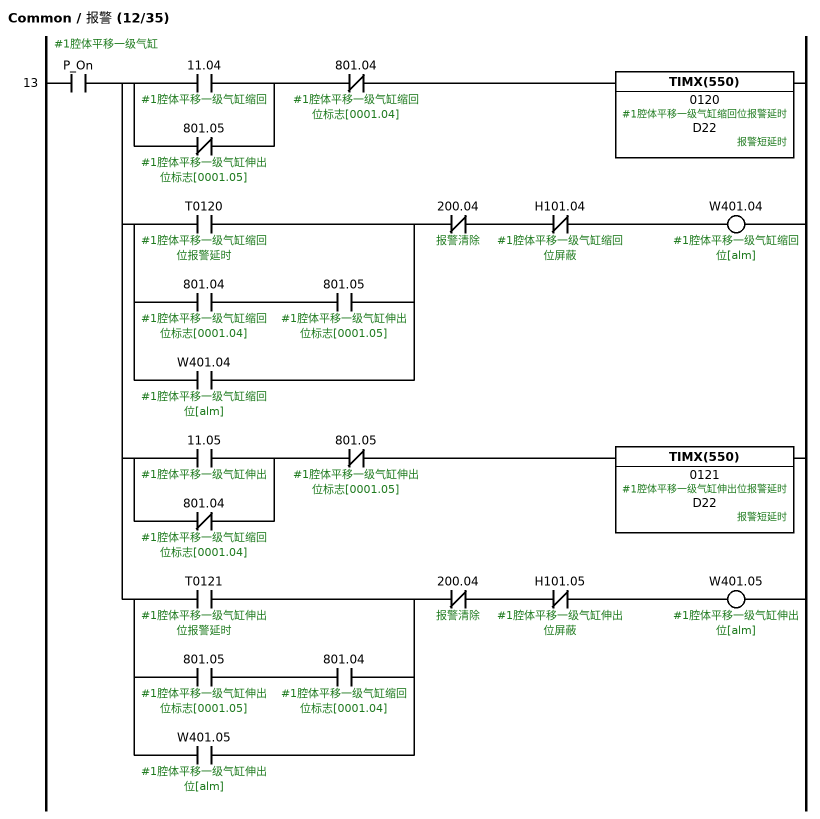
; rung 13: #1腔体平移一级气缸
LD P_On
OUT TR0
LD 11.04  ; #1腔体平移一级气缸缩回
ORNOT 801.05  ; #1腔体平移一级气缸伸出位标志[0001.05]
ANDLD
ANDNOT 801.04  ; #1腔体平移一级气缸缩回位标志[0001.04]
TIMX(550) 0120 D22  ; 报警短延时, #1腔体平移一级气缸缩回位报警延时
LD TR0
LD T0120  ; #1腔体平移一级气缸缩回位报警延时
LD 801.04  ; #1腔体平移一级气缸缩回位标志[0001.04]
AND 801.05  ; #1腔体平移一级气缸伸出位标志[0001.05]
ORLD
OR W401.04  ; #1腔体平移一级气缸缩回位[alm]
ANDLD
ANDNOT 200.04  ; 报警清除
ANDNOT H101.04  ; #1腔体平移一级气缸缩回位屏蔽
OUT W401.04  ; #1腔体平移一级气缸缩回位[alm]
LD TR0
LD 11.05  ; #1腔体平移一级气缸伸出
ORNOT 801.04  ; #1腔体平移一级气缸缩回位标志[0001.04]
ANDLD
ANDNOT 801.05  ; #1腔体平移一级气缸伸出位标志[0001.05]
TIMX(550) 0121 D22  ; 报警短延时, #1腔体平移一级气缸伸出位报警延时
LD TR0
LD T0121  ; #1腔体平移一级气缸伸出位报警延时
LD 801.05  ; #1腔体平移一级气缸伸出位标志[0001.05]
AND 801.04  ; #1腔体平移一级气缸缩回位标志[0001.04]
ORLD
OR W401.05  ; #1腔体平移一级气缸伸出位[alm]
ANDLD
ANDNOT 200.04  ; 报警清除
ANDNOT H101.05  ; #1腔体平移一级气缸伸出位屏蔽
OUT W401.05  ; #1腔体平移一级气缸伸出位[alm]

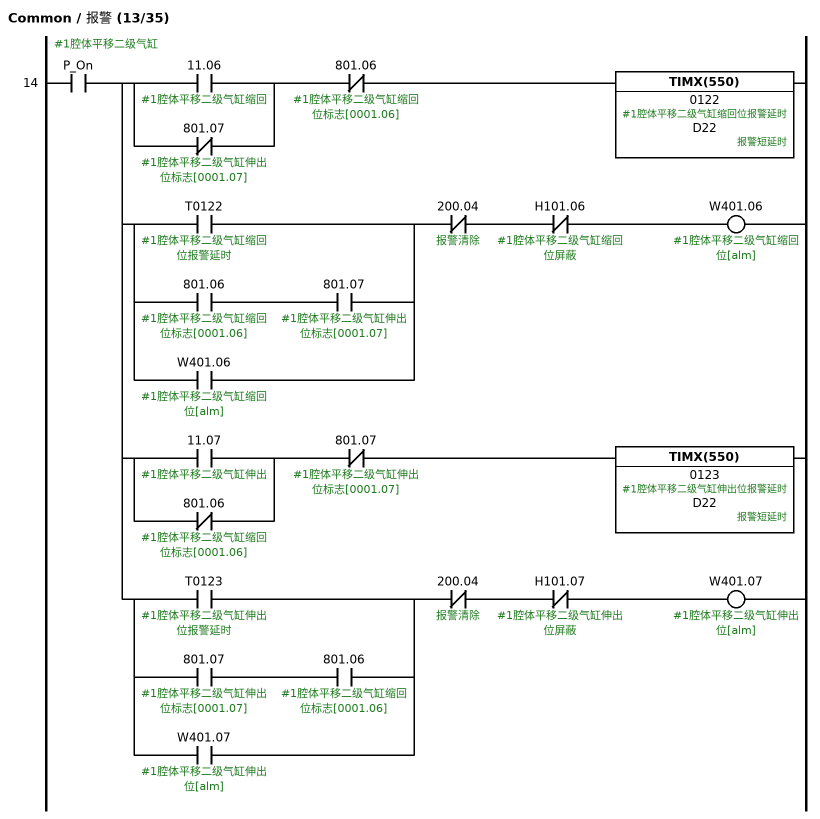
; rung 14: #1腔体平移二级气缸
LD P_On
OUT TR0
LD 11.06  ; #1腔体平移二级气缸缩回
ORNOT 801.07  ; #1腔体平移二级气缸伸出位标志[0001.07]
ANDLD
ANDNOT 801.06  ; #1腔体平移二级气缸缩回位标志[0001.06]
TIMX(550) 0122 D22  ; 报警短延时, #1腔体平移二级气缸缩回位报警延时
LD TR0
LD T0122  ; #1腔体平移二级气缸缩回位报警延时
LD 801.06  ; #1腔体平移二级气缸缩回位标志[0001.06]
AND 801.07  ; #1腔体平移二级气缸伸出位标志[0001.07]
ORLD
OR W401.06  ; #1腔体平移二级气缸缩回位[alm]
ANDLD
ANDNOT 200.04  ; 报警清除
ANDNOT H101.06  ; #1腔体平移二级气缸缩回位屏蔽
OUT W401.06  ; #1腔体平移二级气缸缩回位[alm]
LD TR0
LD 11.07  ; #1腔体平移二级气缸伸出
ORNOT 801.06  ; #1腔体平移二级气缸缩回位标志[0001.06]
ANDLD
ANDNOT 801.07  ; #1腔体平移二级气缸伸出位标志[0001.07]
TIMX(550) 0123 D22  ; 报警短延时, #1腔体平移二级气缸伸出位报警延时
LD TR0
LD T0123  ; #1腔体平移二级气缸伸出位报警延时
LD 801.07  ; #1腔体平移二级气缸伸出位标志[0001.07]
AND 801.06  ; #1腔体平移二级气缸缩回位标志[0001.06]
ORLD
OR W401.07  ; #1腔体平移二级气缸伸出位[alm]
ANDLD
ANDNOT 200.04  ; 报警清除
ANDNOT H101.07  ; #1腔体平移二级气缸伸出位屏蔽
OUT W401.07  ; #1腔体平移二级气缸伸出位[alm]

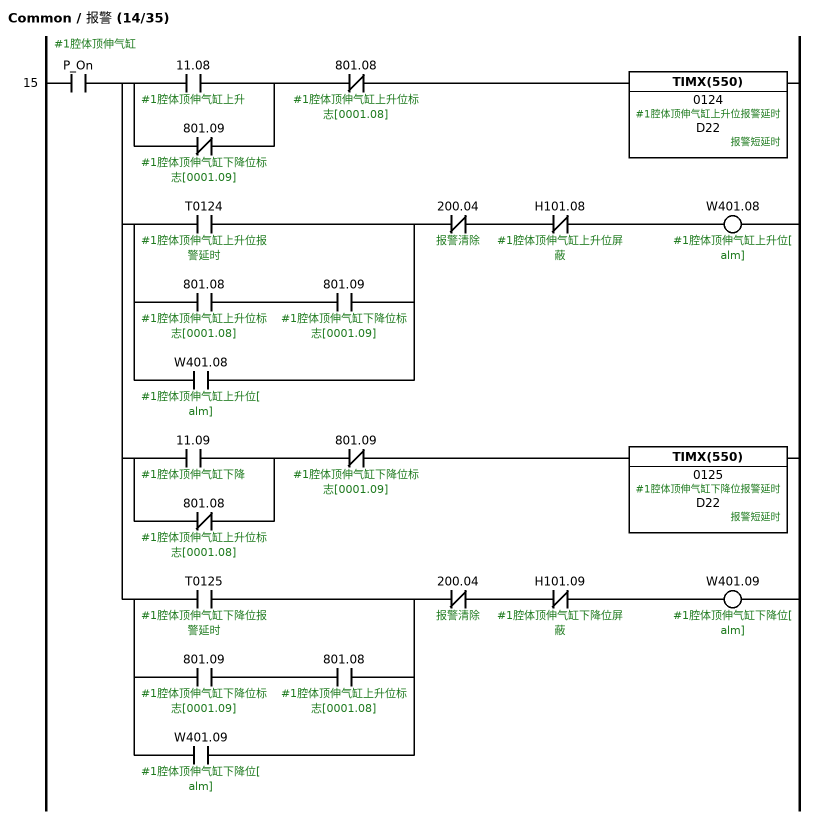
; rung 15: #1腔体顶伸气缸
LD P_On
OUT TR0
LD 11.08  ; #1腔体顶伸气缸上升
ORNOT 801.09  ; #1腔体顶伸气缸下降位标志[0001.09]
ANDLD
ANDNOT 801.08  ; #1腔体顶伸气缸上升位标志[0001.08]
TIMX(550) 0124 D22  ; 报警短延时, #1腔体顶伸气缸上升位报警延时
LD TR0
LD T0124  ; #1腔体顶伸气缸上升位报警延时
LD 801.08  ; #1腔体顶伸气缸上升位标志[0001.08]
AND 801.09  ; #1腔体顶伸气缸下降位标志[0001.09]
ORLD
OR W401.08  ; #1腔体顶伸气缸上升位[alm]
ANDLD
ANDNOT 200.04  ; 报警清除
ANDNOT H101.08  ; #1腔体顶伸气缸上升位屏蔽
OUT W401.08  ; #1腔体顶伸气缸上升位[alm]
LD TR0
LD 11.09  ; #1腔体顶伸气缸下降
ORNOT 801.08  ; #1腔体顶伸气缸上升位标志[0001.08]
ANDLD
ANDNOT 801.09  ; #1腔体顶伸气缸下降位标志[0001.09]
TIMX(550) 0125 D22  ; 报警短延时, #1腔体顶伸气缸下降位报警延时
LD TR0
LD T0125  ; #1腔体顶伸气缸下降位报警延时
LD 801.09  ; #1腔体顶伸气缸下降位标志[0001.09]
AND 801.08  ; #1腔体顶伸气缸上升位标志[0001.08]
ORLD
OR W401.09  ; #1腔体顶伸气缸下降位[alm]
ANDLD
ANDNOT 200.04  ; 报警清除
ANDNOT H101.09  ; #1腔体顶伸气缸下降位屏蔽
OUT W401.09  ; #1腔体顶伸气缸下降位[alm]

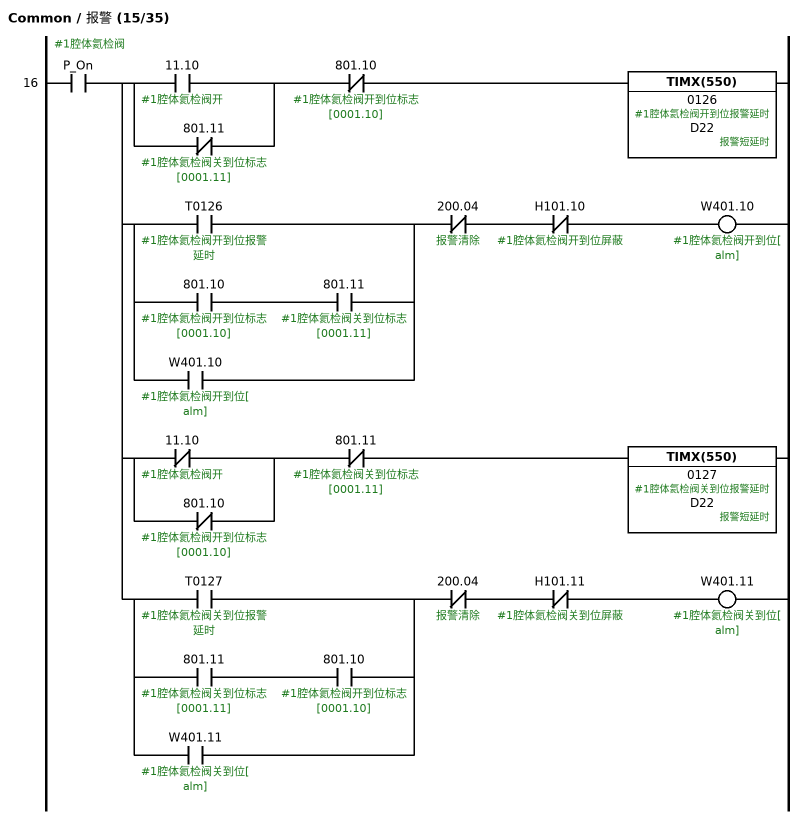
; rung 16: #1腔体氦检阀
LD P_On
OUT TR0
LD 11.10  ; #1腔体氦检阀开
ORNOT 801.11  ; #1腔体氦检阀关到位标志[0001.11]
ANDLD
ANDNOT 801.10  ; #1腔体氦检阀开到位标志[0001.10]
TIMX(550) 0126 D22  ; 报警短延时, #1腔体氦检阀开到位报警延时
LD TR0
LD T0126  ; #1腔体氦检阀开到位报警延时
LD 801.10  ; #1腔体氦检阀开到位标志[0001.10]
AND 801.11  ; #1腔体氦检阀关到位标志[0001.11]
ORLD
OR W401.10  ; #1腔体氦检阀开到位[alm]
ANDLD
ANDNOT 200.04  ; 报警清除
ANDNOT H101.10  ; #1腔体氦检阀开到位屏蔽
OUT W401.10  ; #1腔体氦检阀开到位[alm]
LD TR0
LDNOT 11.10  ; #1腔体氦检阀开
ORNOT 801.10  ; #1腔体氦检阀开到位标志[0001.10]
ANDLD
ANDNOT 801.11  ; #1腔体氦检阀关到位标志[0001.11]
TIMX(550) 0127 D22  ; 报警短延时, #1腔体氦检阀关到位报警延时
LD TR0
LD T0127  ; #1腔体氦检阀关到位报警延时
LD 801.11  ; #1腔体氦检阀关到位标志[0001.11]
AND 801.10  ; #1腔体氦检阀开到位标志[0001.10]
ORLD
OR W401.11  ; #1腔体氦检阀关到位[alm]
ANDLD
ANDNOT 200.04  ; 报警清除
ANDNOT H101.11  ; #1腔体氦检阀关到位屏蔽
OUT W401.11  ; #1腔体氦检阀关到位[alm]

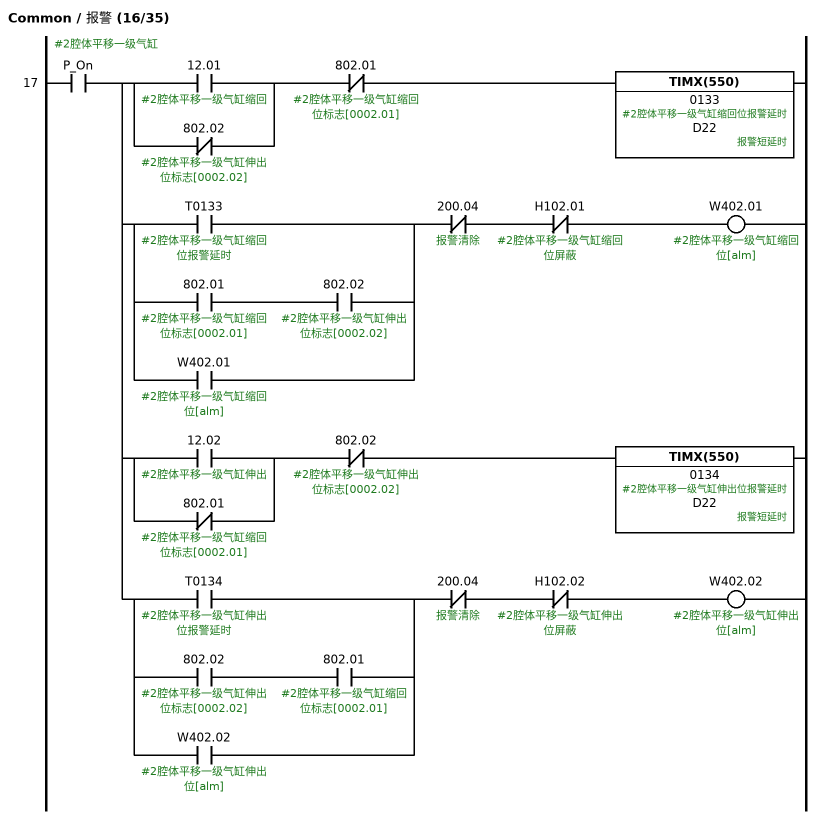
; rung 17: #2腔体平移一级气缸
LD P_On
OUT TR0
LD 12.01  ; #2腔体平移一级气缸缩回
ORNOT 802.02  ; #2腔体平移一级气缸伸出位标志[0002.02]
ANDLD
ANDNOT 802.01  ; #2腔体平移一级气缸缩回位标志[0002.01]
TIMX(550) 0133 D22  ; 报警短延时, #2腔体平移一级气缸缩回位报警延时
LD TR0
LD T0133  ; #2腔体平移一级气缸缩回位报警延时
LD 802.01  ; #2腔体平移一级气缸缩回位标志[0002.01]
AND 802.02  ; #2腔体平移一级气缸伸出位标志[0002.02]
ORLD
OR W402.01  ; #2腔体平移一级气缸缩回位[alm]
ANDLD
ANDNOT 200.04  ; 报警清除
ANDNOT H102.01  ; #2腔体平移一级气缸缩回位屏蔽
OUT W402.01  ; #2腔体平移一级气缸缩回位[alm]
LD TR0
LD 12.02  ; #2腔体平移一级气缸伸出
ORNOT 802.01  ; #2腔体平移一级气缸缩回位标志[0002.01]
ANDLD
ANDNOT 802.02  ; #2腔体平移一级气缸伸出位标志[0002.02]
TIMX(550) 0134 D22  ; 报警短延时, #2腔体平移一级气缸伸出位报警延时
LD TR0
LD T0134  ; #2腔体平移一级气缸伸出位报警延时
LD 802.02  ; #2腔体平移一级气缸伸出位标志[0002.02]
AND 802.01  ; #2腔体平移一级气缸缩回位标志[0002.01]
ORLD
OR W402.02  ; #2腔体平移一级气缸伸出位[alm]
ANDLD
ANDNOT 200.04  ; 报警清除
ANDNOT H102.02  ; #2腔体平移一级气缸伸出位屏蔽
OUT W402.02  ; #2腔体平移一级气缸伸出位[alm]

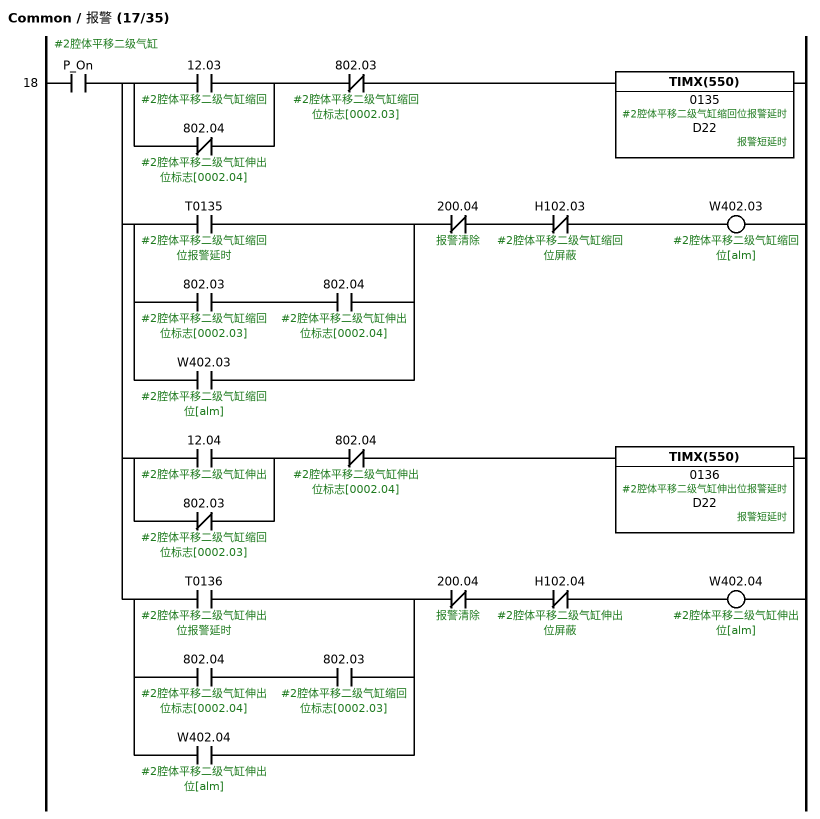
; rung 18: #2腔体平移二级气缸
LD P_On
OUT TR0
LD 12.03  ; #2腔体平移二级气缸缩回
ORNOT 802.04  ; #2腔体平移二级气缸伸出位标志[0002.04]
ANDLD
ANDNOT 802.03  ; #2腔体平移二级气缸缩回位标志[0002.03]
TIMX(550) 0135 D22  ; 报警短延时, #2腔体平移二级气缸缩回位报警延时
LD TR0
LD T0135  ; #2腔体平移二级气缸缩回位报警延时
LD 802.03  ; #2腔体平移二级气缸缩回位标志[0002.03]
AND 802.04  ; #2腔体平移二级气缸伸出位标志[0002.04]
ORLD
OR W402.03  ; #2腔体平移二级气缸缩回位[alm]
ANDLD
ANDNOT 200.04  ; 报警清除
ANDNOT H102.03  ; #2腔体平移二级气缸缩回位屏蔽
OUT W402.03  ; #2腔体平移二级气缸缩回位[alm]
LD TR0
LD 12.04  ; #2腔体平移二级气缸伸出
ORNOT 802.03  ; #2腔体平移二级气缸缩回位标志[0002.03]
ANDLD
ANDNOT 802.04  ; #2腔体平移二级气缸伸出位标志[0002.04]
TIMX(550) 0136 D22  ; 报警短延时, #2腔体平移二级气缸伸出位报警延时
LD TR0
LD T0136  ; #2腔体平移二级气缸伸出位报警延时
LD 802.04  ; #2腔体平移二级气缸伸出位标志[0002.04]
AND 802.03  ; #2腔体平移二级气缸缩回位标志[0002.03]
ORLD
OR W402.04  ; #2腔体平移二级气缸伸出位[alm]
ANDLD
ANDNOT 200.04  ; 报警清除
ANDNOT H102.04  ; #2腔体平移二级气缸伸出位屏蔽
OUT W402.04  ; #2腔体平移二级气缸伸出位[alm]

